      U     "MAL1S022Par".Par.FlagProcess2.Turning1WithoutSpraying;
      U     "MAL1S022Par".Par.FlagFunction_1.TurningStart;
      UN    "G205M".A_2611_MXZ41MA.Ma.StAdjusted; // target position turning reached
      FP    "MAL1S022Par".Par.FlagProcess2.StartFirstTurningFP;
      =     "MAL1S022Par".Par.FlagProcess2.StartFirstDosingFP;
      S     "MAL1S022Par".Par.FlagProcess2.StartFirstTurningRound;

      U     "MAL1S022Par".Par.FlagProcess2.StartFirstDosingFP;
      U     "MAL1S022Par".Par.FlagProcess2.StartFirstTurningFP;
      SPB   trn1;
      L     "MAL1S022Par".Par.ParIntMachine.ActualStep;
      T     "MAL1S022Par".Par.ParIntProcess.PrevStep1stTurn;
trn1: NOP   0;

      U     "G205M".A_2611_MXZ41MA.Ma.StAdjusted; // target position turning reached
      O(    ;
      L     "MAL1S022Par".ActTimeStepProcess.StepTimeActHourTotal; // Steptime in hours overall
      L     "MAL1S022Par".StepAct.StartTurningRound_1;
      >I    ;
      U(    ;
      O     "G205M".A_2611_MXZ41MA.Ma.OutAdjusted; // target position turning reached
      O(    ;
      UN    "G205M".A_2611_BZS46.StTrue; // stop fan side
      U     "G205M".A_2611_BZS44.StTrue; // stop discharge side
      U     "MAL1S022Par".Par.FlagFunction_1.TurningRight;
      )     ;
      O(    ;
      U     "G205M".A_2611_BZS46.StTrue; // stop fan side
      UN    "G205M".A_2611_BZS44.StTrue; // stop discharge side
      U     "MAL1S022Par".Par.FlagFunction_1.TurningLeft;
      )     ;
      )     ;
      )     ;
      O(    ;
      L     "MAL1S022Par".StepAct.StartTurningRound_1;
      L     0;
      <D    ; // negative, no turning 1
      )     ;
      U     "MAL1S022Par".Par.FlagProcess2.StartFirstTurningRound;
      R     "MAL1S022Par".Par.FlagProcess2.StartFirstTurningRound;
      R     "MAL1S022Par".Par.Switches1.StaOn08; // Turning1WithSpraying
      R     "MAL1S022Par".Par.Switches1.StaOn09; // Turning1WithDosing

// turning 2
      UN    "MAL1S022Par".Par.FlagProcess2.StartFirstTurningRound; // Unsinnige Rezeptwerte
      U(    ;
      L     1;
      L     "MAL1S022Par".StepAct.StartTurningRound_2;
      <>I   ;
      )     ;
      U(    ;
      O(    ; // Nach Rezept
      L     "MAL1S022Par".ActTimeStepProcess.StepTimeActHourTotal; // Steptime in hours overall
      L     "MAL1S022Par".StepAct.StartTurningRound_2;
      ==I   ;
      UN    "G205M".A_2611_MXZ41MA.Ma.StAdjusted; // target position turning reached
      )     ;
      O(    ; // Selbsthaltung
      L     "MAL1S022Par".ActTimeStepProcess.StepTimeActHourTotal; // Steptime in hours overall
      L     "MAL1S022Par".StepAct.StartTurningRound_2;
      <>I   ;
      U     "MAL1S022Par".Par.FlagProcess2.StartSecondTurningRound;
      )     ;
      )     ;
      S     "MAL1S022Par".Par.FlagProcess2.Turning2WithoutSpraying;
      S     "MAL1S022Par".Par.FlagFunction_1.TurningStart;
// turning 2 with spraying
      U(    ;
      L     1;
      L     "MAL1S022Par".StepAct.TurningWithSpraying_2;
      ==I   ;
      U(    ;
      L     "MAL1S022Par".Par.ParIntMachine.ActualStep;
      L     "MAL1S022Par".Par.ParIntProcess.PrevStep2ndTurn;
      ==I   ;
      )     ;
      )     ;
      O(    ;
      L     "MAL1S022Par".Par.ParIntMachine.ActualStep;
      L     "MAL1S022Par".Par.ParIntProcess.PrevStep2ndTurn;
      <>I   ;
      U     "MAL1S022Par".Par.Switches1.StaOn10; // Turning2WithSpraying
      )     ;
      U     "MAL1S022Par".Par.FlagProcess2.Turning2WithoutSpraying;
      S     "MAL1S022Par".Par.FlagProcess2.Turning2WithSpraying;
// turning 2 with spraying and GA3
      U(    ;
      L     1;
      L     "MAL1S022Par".StepAct.TurningWithDosing_2;
      ==I   ; // turning 2 with spraying and GA3 on
      U(    ;
      L     "MAL1S022Par".Par.ParIntMachine.ActualStep;
      L     "MAL1S022Par".Par.ParIntProcess.PrevStep2ndTurn;
      ==I   ;
      )     ;
      )     ;
      O(    ;
      L     "MAL1S022Par".Par.ParIntMachine.ActualStep;
      L     "MAL1S022Par".Par.ParIntProcess.PrevStep2ndTurn;
      <>I   ;
      U     "MAL1S022Par".Par.Switches1.StaOn11; // Turning2WithDosing
      )     ;
      U     "MAL1S022Par".Par.FlagProcess2.Turning2WithoutSpraying;
      S     "MAL1S022Par".Par.FlagProcess2.Turning2WithSpraying;
      S     "MAL1S022Par".Par.FlagProcess2.Turning2WithDosing;

      U     "MAL1S022Par".Par.FlagProcess2.Turning2WithoutSpraying;
      U     "MAL1S022Par".Par.FlagFunction_1.TurningStart;
      UN    "G205M".A_2611_MXZ41MA.Ma.StAdjusted; // target position turning reached
      FP    "MAL1S022Par".Par.FlagProcess2.StartSecondTurningFP;
      =     "MAL1S022Par".Par.FlagProcess2.StartSecondDosingFP;
      S     "MAL1S022Par".Par.FlagProcess2.StartSecondTurningRound;

      U     "MAL1S022Par".Par.FlagProcess2.StartSecondDosingFP;
      U     "MAL1S022Par".Par.FlagProcess2.StartSecondTurningFP;
      SPB   trn2;
      L     "MAL1S022Par".Par.ParIntMachine.ActualStep;
      T     "MAL1S022Par".Par.ParIntProcess.PrevStep2ndTurn;
trn2: NOP   0;

      U     "G205M".A_2611_MXZ41MA.Ma.StAdjusted; // target position turning reached
      O(    ;
      L     "MAL1S022Par".ActTimeStepProcess.StepTimeActHourTotal; // Steptime in hours overall
      L     "MAL1S022Par".StepAct.StartTurningRound_2;
      >I    ;
      U(    ;
      O     "G205M".A_2611_MXZ41MA.Ma.OutAdjusted; // target position turning reached
      O(    ;
      UN    "G205M".A_2611_BZS46.StTrue; // stop fan side
      U     "G205M".A_2611_BZS44.StTrue; // stop discharge side
      U     "MAL1S022Par".Par.FlagFunction_1.TurningRight;
      )     ;
      O(    ;
      U     "G205M".A_2611_BZS46.StTrue; // stop fan side
      UN    "G205M".A_2611_BZS44.StTrue; // stop discharge side
      U     "MAL1S022Par".Par.FlagFunction_1.TurningLeft;
      )     ;
      )     ;
      )     ;
      O(    ;
      L     "MAL1S022Par".StepAct.StartTurningRound_2;
      L     0;
      <D    ; // negative, no turning 2
      )     ;
      U     "MAL1S022Par".Par.FlagProcess2.StartSecondTurningRound;
      R     "MAL1S022Par".Par.FlagProcess2.StartSecondTurningRound;
      R     "MAL1S022Par".Par.Switches1.StaOn10; // Turning2WithSpraying
      R     "MAL1S022Par".Par.Switches1.StaOn11; // Turning2WithDosing

      L     3600;
      T     "MAL1S022Par".Par.ParIntMachine.TargetPosTravDriTurnRigt; // 360° = endposition turning right

// find turning direction spez. APU: right ==> forward, left ==> reverse
      U     "MAL1S022Par".Par.FlagGen.TurningStarted;
      O(    ;
      UN    "MAL1S022Par".Par.FlagProcess2.Turning1WithoutSpraying;
      UN    "MAL1S022Par".Par.FlagProcess2.Turning2WithoutSpraying;
      )     ;
      SPB   tuen;
      L     "MAL1S022Par".Par.ParIntMachine.TargetPosTravDriTurnRigt; // 360° = endposition turning right
      T     "G205M".A_2611_MXZ41MA.Ma.InPositionTarget; // target position turning

      U(    ;
      L     "G205M".A_2611_MXZ41MA.Ma.OutPositionAngle;
      L     1800;
      <I    ; // condition turning right (clockwise)
      )     ;
      O     "G205M".A_2611_BZS46.StTrue; // stop fan side
      UN    "G205M".A_2611_BZS44.StTrue; // stop discharge side
      S     "MAL1S022Par".Par.FlagFunction_1.TurningRight;
      S     "MAL1S022Par".Par.FlagGen.TurningStarted;
      SPB   E603;
      L     "MAL1S022Par".Par.ParIntMachine.TargetPosTravDriTurnLeft; // 0° = endposition turning left
      T     "G205M".A_2611_MXZ41MA.Ma.InPositionTarget; // target position turning

      U(    ;
      L     "G205M".A_2611_MXZ41MA.Ma.OutPositionAngle;
      L     1800;
      >=I   ; // condition turning left (counterclockwise)
      )     ;
      O     "G205M".A_2611_BZS44.StTrue; // stop discharge side
      UN    "G205M".A_2611_BZS46.StTrue; // stop fan side
      S     "MAL1S022Par".Par.FlagFunction_1.TurningLeft;
      S     "MAL1S022Par".Par.FlagGen.TurningStarted;
      SPB   E603;
tuen: NOP   0;

// reset turning right (clockwise)
      U     "MAL1S022Par".Par.FlagFunction_1.TurningRight;
      U(    ;
//      O     "G202M"._2111_MXZ41MA.Ma.StAdjusted    // target position turning reached
      O(    ;
      L     "G205M".A_2611_MXZ41MA.Ma.OutPositionAngle;
      L     "G205M".A_2611_MXZ41MA.Ma.Par.ParTolPosition;
      +I    ;
      L     "MAL1S022Par".Par.ParIntMachine.TargetPosTravDriTurnRigt;
      >=I   ;
      )     ;
      O     "G205M".A_2611_BZS44.StTrue; // stop discharge side
      )     ;
      R     "MAL1S022Par".Par.FlagFunction_1.TurningRight;
      R     "MAL1S022Par".Par.FlagFunction_1.TurningStart;

// reset turning left (counterclockwise)
      U     "MAL1S022Par".Par.FlagFunction_1.TurningLeft;
      U(    ;
//      O     "G202M"._2111_MXZ41MA.Ma.StAdjusted    // target position turning reached
      O(    ;
      L     "G205M".A_2611_MXZ41MA.Ma.OutPositionAngle;
      L     "G205M".A_2611_MXZ41MA.Ma.Par.ParTolPosition;
      -I    ;
      L     "MAL1S022Par".Par.ParIntMachine.TargetPosTravDriTurnLeft;
      <=I   ;
      )     ;
      O     "G205M".A_2611_BZS46.StTrue; // stop fan side
      )     ;
      R     "MAL1S022Par".Par.FlagFunction_1.TurningLeft;
      R     "MAL1S022Par".Par.FlagFunction_1.TurningStart;

// - Case of fast speed to protect a 2nd start during same hours as finsihed
      U     "MAL1S022Par".Par.FlagGen.TurningStarted;
      UN    "MAL1S022Par".Par.FlagProcess.ProcessEnd; // JV210808 to finish last turning
      UN    "MAL1S022StepValues".StartStep; // start step for average calculating
      U(    ;
      O(    ; // Nach Rezept
      L     "MAL1S022Par".ActTimeStepProcess.StepTimeActHourTotal; // Steptime in hours overall
      L     "MAL1S022Par".StepAct.StartTurningRound_1;
      <=I   ; // JV 250808
      UN    "MAL1S022Par".Par.FlagProcess2.StartFirstTurningRound; // JV 250808
      )     ;
      O(    ; // Nach Rezept
      L     "MAL1S022Par".ActTimeStepProcess.StepTimeActHourTotal; // Steptime in hours overall
      L     "MAL1S022Par".StepAct.StartTurningRound_2;
      <=I   ; // JV 250808
      UN    "MAL1S022Par".Par.FlagProcess2.StartSecondTurningRound; // JV 250808
      )     ;
      )     ;
      O(    ;
      UN    "G205M".A_2611_MXZ41MA.Ma.OutAdjusted; // target position turning reached
      UN    "MAL1S022Par".Par.FlagFunction_1.StepUnloading;
      )     ;
      SPB   e603;

// reset turning flag
      U     "MAL1S022Par".Par.FlagGen.TurningStarted;
      ON    "MAL1S022Par".Par.FlagProcess.ProcessActive;
      R     "MAL1S022Par".Par.FlagGen.TurningStarted;
      R     "MAL1S022Par".Par.FlagProcess2.Turning1WithoutSpraying;
      R     "MAL1S022Par".Par.FlagProcess2.Turning2WithoutSpraying;
      R     "MAL1S022Par".Par.FlagProcess2.Turning1WithSpraying;
      R     "MAL1S022Par".Par.FlagProcess2.Turning2WithSpraying;
      R     "MAL1S022Par".Par.FlagProcess2.Turning1WithDosing;
      R     "MAL1S022Par".Par.FlagProcess2.Turning2WithDosing;
      R     "MAL1S022Par".Par.FlagFunction_1.TurningStart;
      R     "MAL1S022Par".Par.FlagProcess2.StartFirstTurningRound; // JV 250808
      R     "MAL1S022Par".Par.FlagProcess2.StartSecondTurningRound; // JV 250808
      SET   ;
      R     "MAL1S022StepValues".StartStep; // start step for average calculating
e630: NOP   0;
      UN    "MAL1S022Par".Par.FlagProcess.ProcessActive;
      R     "MAL1S022Par".Par.FlagProcess2.StartFirstTurningRound;
      R     "MAL1S022Par".Par.FlagProcess2.StartSecondTurningRound;
      R     "MAL1S022Par".Par.Switches1.StaOn08; // Turning1WithSpraying
      R     "MAL1S022Par".Par.Switches1.StaOn09; // Turning1WithDosing
      R     "MAL1S022Par".Par.Switches1.StaOn10; // Turning2WithSpraying
      R     "MAL1S022Par".Par.Switches1.StaOn11; // Turning2WithDosing

      L     "G205M".A_2611_MXZ41MA.Ma.OutPositionAngle;
      T     "G205M".A_2611_MXZ41MA.Ma.OutPositionAngle;

      L     "G205M".A_2611_MXZ41MA.Ma.OutPositionRel;
      T     "G205M".A_2611_MXZ41MA.Ma.OutPositionRel;

e603: NOP   0;
E603: NOP   0;


NETWORK
TITLE =ASW_6040: Set fanspeed by delta-t
//Die Drehzahl des Ventilators wird zwischen dem Rezeptsollwert, als Untere
//Grenze, und 100% oder Rezeptsollwert, als obere Grenze, geregelt. Die Regelung
//erfolgt nach folgendem Prinzip:
//"Delta-T" ist die Differenz zwischen der Soll-Temperatur (Rezeptsollwert) unter
//der Horde und der gemessenen Ist-Temperatur über der Horde.
//Steigt die Ist-Temperatur über der Horde und "Delta-T" wird > als der Sollwert
//im Rezept, so wird die Drehzahl des Ventilators stufenweise erhöht. Maximale
//Drehzahl ist 100% oder Rezeptsollwert.
//Sinkt die Ist-Temperatur über der Horde und "Delta-T" wird < als der Sollwert
//im
//Rezept, so wird die Drehzahl des Ventilators stufenweise verringert. Minimale
//Drehzahl ist der Rezeptsollwert.
//Die Rampen (Stufen) werden durch den Technologen festgelegt und in Programmcode
//eingetragen. Es sind keine Rezeptsollwerte.
      NOP   0;
// recipe setpoint
      L     "MAL1S022Par".StepAct.SpeedVentilatorBasic;
      L     0;
      ==I   ; // no fan during turning
      SPB   e604; // JV040908
      L     "MAL1S022Par".Par.ProcessValue.StepTimeAct; // in ms
      L     L#1000; // in first secunde steptime
      >D    ;
      SPB   regu;
      SPA   Summ;
regu: NOP   0;

      U     "MAL1S022".ToASW.CmdModify;
      SPB   Summ;

// Setpoint
      L     "MAL1S022Par".StepAct.TemperaturAboveFloor;
      L     "MAL1S022Par".StepAct.TemperaturBelowFloor;
      -D    ;
      T     "MAL1S022Par".Par.ProcessValue.SetpointDeltaTempDint;
// actual value
      L     "G208M".A_2691_BTE02.OutValueUnits; //AIR TEMPERATURE ABOVE FLOOR
      L     "G208M".A_2691_BTE01.OutValueUnits; //AIR TEMPERATURE BELOW FLOOR
      -D    ;
      T     "MAL1S022Par".Par.ProcessValue.ActValueDeltaTempDint;
// flags to inc/dec
      L     "MAL1S022Par".Par.ProcessValue.SetpointDeltaTempDint;
      -D    ;
      T     "MAL1S022Par".Par.ProcessValue.ResultDeltaTemp;
      L     L#0;
      >D    ;
      =     "MAL1S022Par".Par.FlagProcess1.DeltaTempPlus;
      <D    ;
      =     "MAL1S022Par".Par.FlagProcess1.DeltaTempMinus;

      U     "MAL1S022Par".Par.FlagProcess1.DeltaTempPlus;
      U     "SYS_Scan0_Tick1min";
      SPBN  dec;
      L     "MAL1S022Par".Par.ParIntMachine.TargetSpeedGermFan;
      L     100; // linmit max
      >=I   ;
      SPB   dec;
      L     "MAL1S022Par".Par.ParIntMachine.TargetSpeedGermFan;
      L     1;
      +I    ;
      T     "MAL1S022Par".Par.ParIntMachine.TargetSpeedGermFan;
      SPA   e604;
dec:  NOP   0;
      U     "MAL1S022Par".Par.FlagProcess1.DeltaTempMinus;
      U     "SYS_Scan0_Tick1min";
      SPBN  e604;
      L     "MAL1S022Par".Par.ParIntMachine.TargetSpeedGermFan;
      L     "MAL1S022Par".StepAct.SpeedVentilatorBasic; // linmit min
      <=I   ;
      SPB   e604;
      L     "MAL1S022Par".Par.ParIntMachine.TargetSpeedGermFan;
      L     1;
      -I    ;
      T     "MAL1S022Par".Par.ParIntMachine.TargetSpeedGermFan;
      SPA   e604;

Summ: NOP   0;
      L     "MAL1S022Par".StepAct.SpeedVentilatorBasic;
      T     "MAL1S022Par".Par.ParIntMachine.TargetSpeedGermFan;
      U     "MAL1S022Par".Par.FlagProcess.ProcessEnd; // JV030908
      UN    "MAL1S022".PCRead.Step.StEmptying;
      UN    "MAL1S022".PCRead.Step.StEmptied;
      SPBN  e604;
      L     "MAL1S022Par".Par.ParIntProcess.SavedTargetSpeedGermFan;
      T     "MAL1S022Par".Par.ParIntMachine.TargetSpeedGermFan;
e604: NOP   0;
// store actual setpoint
      U     "MAL1S022Par".Par.FlagProcess.ProcessActive;
      U(    ;
      L     "MAL1S022Par".StepAct.SpeedVentilatorBasic;
      L     0; // setpoint recipe > 0
      >I    ;
      )     ;
      SPBN  E604;
      L     "MAL1S022Par".StepAct.SpeedVentilatorBasic;
      T     "MAL1S022Par".Par.ParIntProcess.SavedTargetSpeedGermFan;
E604: NOP   0;

NETWORK
TITLE =ASW_6050: Position waste air
//Der Betriebsart Sommerbetrieb/Winterbetrieb wird durch den Bediener per Rezept
//bestimmt.
//Wird die Kühlung im Rezept angewählt, so erfolgt die Umschaltung AUF
//Sommerbetrieb. Die Frischluftklappe wird nach dem Rezeptsollwert gestellt.
//Es erfolgt keine Regelung.
//Wird die Kühlung im Rezept abgewählt, so erfolgt die Umschaltung AUF
//Winterbetrieb. Die Frischluftklappe wird zuerst nach dem Rezeptsollwert
//gestellt. Der Rezeptsollwert ist die untere Grenze für die Regelung.
//Wird die Soll-Temperatur unter der Horde von Kühl- Heizanlage nicht eingehalten
//-Temperatur zu hoch und der Schaltpunkt überschritten, so wird die
//Frischluftklappe stufenweise geöffnet.
//Maximalwert ist 100%.
//Wird die Soll-Temperatur unter der Horde von Kühl- Heizanlage nicht eingehalten
//-Temperatur zu niedrig und der Schaltpunkt unterschritten, so wird die
//Frischluftklappe stufenweise geschlossen.
//Minimalwert ist der Rezeptsollwert.
      NOP   0;
// setpoint waste air                    = 100% - setpoint fresh air
      L     100;
      L     "MAL1S022Par".StepAct.PosFreshAirFlapBasic;
      -I    ;
      T     "MAL1S022Par".StepAct.PosWasteAirFlapBasic;

// setpoint limit maximal position fresh air
      L     100;
      T     "MAL1S022Par".StepAct.PosFreshAirFlapMax; // limit max
      L     L#10; // 1,0°
      T     "MAL1S022Par".StepAct.DeltaTempSwitchpointAir;

// recipe setpoint
      L     "MAL1S022Par".Par.ProcessValue.StepTimeAct; // in ms
      L     L#1000; // in first secunde steptime
      >D    ;
      SPB   Reg;
      SPA   summ;
Reg:  NOP   0;

// Cooling or heating from cooling defive active --> no flap regulation!
//      U     "ENG_RemarkFlag"
//      U     "ComDB_Cooling".Ma.ACK.ActivFlag.Cool.Germinating_1_Started // Internal or external coooling is running
//      O     "MAL1S017".ToASW.CmdModify
//      SPB   summ

//Conditions to activate cooling -- With flap regulation
      U(    ;
      L     1;
      L     "MAL1S022Par".StepAct.Cooling; // On/Off
      ==I   ; // Cooling on
      U     "MAL1S022Par".Par.FlagProcess.ProcessActive;
      )     ;
      U     "G210M".A_2660_MXZ01.StStartedFwd;
      U     "G210M".A_2660_MXZ02.StStartedFwd;
      U(    ;
      L     "G269M".A_3191_BTE11.OutValueUnits; //WET BULB TEMPERATURE OUTSIDE
      L     20; // 2,0°C Hysteresis
      -D    ;
      L     "MAL1S022Par".StepAct.TemperaturBelowFloor; //SET POINT TEMPERATURE RECIPE
      >=D   ;
      )     ;
      U(    ;
      L     "G208M".A_2691_BTE01.OutValueUnits; //AIR TEMPERATURE BELOW FLOOR GM2
      L     10; // 1,0°C Hysteresis
      -D    ;
      L     "MAL1S022Par".StepAct.TemperaturBelowFloor; //SET POINT TEMPERATURE RECIPE
      >=D   ;
      )     ;
      U(    ;
      L     "G208M".A_2691_BTE02.OutValueUnits; //AIR TEMPERATURE ABOVE FLOOR GM2
      L     20; // 2,0°C Hysteresis
      -D    ;
      L     "MAL1S022Par".StepAct.TemperaturBelowFloor; //SET POINT TEMPERATURE RECIPE
      >=D   ;
      )     ;
      S     "MAL1S022Par".Par.FlagProcess.Cooling_Activ;

      U(    ;
      L     0;
      L     "MAL1S022Par".StepAct.Cooling; // On/Off
      ==I   ; // Cooling off
      )     ;
      ON    "G210M".A_2660_MXZ01.StStartedFwd;
      ON    "G210M".A_2660_MXZ02.StStartedFwd;
      O(    ;
      L     "G269M".A_3191_BTE11.OutValueUnits; //WET BULB TEMPERATURE OUTSIDE
      L     10; // 1,0°C Hysteresis
      +D    ;
      L     "MAL1S022Par".StepAct.TemperaturBelowFloor; //SET POINT TEMPERATURE RECIPE
      <D    ;
      )     ;
      O(    ;
      L     "G208M".A_2691_BTE02.OutValueUnits; //AIR TEMPERATURE ABOVE FLOOR GM1
      L     10; // 1,0°C Hysteresis
      +D    ;
      L     "MAL1S022Par".StepAct.TemperaturBelowFloor; //SET POINT TEMPERATURE RECIPE
      <D    ;
      )     ;
      R     "MAL1S022Par".Par.FlagProcess.Cooling_Activ;

      U     "MAL1S022Par".Par.FlagProcess.Cooling_Activ;
      SPB   summ;

// Check the minimum opening of fresh air louver
      U(    ;
      L     "MAL1S022Par".Par.ParIntMachine.TargetPosFreshAir;
      L     "MAL1S022Par".StepAct.PosFreshAirFlapBasic;
      <I    ;
      )     ;
      SPBN  modi;
      L     "MAL1S022Par".StepAct.PosFreshAirFlapBasic; //Basic position %
      T     "MAL1S022Par".Par.ParIntMachine.TargetPosFreshAir;
modi: NOP   0;

//-Recipe modify-
      U(    ; // Nach gesundem Menschenverstand
      L     "MAL1S022Par".StepAct.PosFreshAirFlapBasic;
      L     "MAL1S022Par".Par.ParIntMachine.TargetPosFreshAir;
      >I    ;
      U     "MAL1S022Par".Par.FlagProcess1.FreshAirFlapOPEN;
      )     ;
      O(    ; // Nach gesundem Menschenverstand
      L     "MAL1S022Par".StepAct.PosFreshAirFlapBasic;
      L     "MAL1S022Par".Par.ParIntMachine.TargetPosFreshAir;
      <I    ;
      U     "MAL1S022Par".Par.FlagProcess1.FreshAirFlapCLOSE;
      )     ;
      O(    ; // Nach gesundem Menschenverstand
      L     "MAL1S022Par".StepAct.PosFreshAirFlapBasic;
      L     "MAL1S022Par".Par.ParIntMachine.TargetPosFreshAir;
      <>I   ;
      UN    "MAL1S022Par".Par.FlagProcess1.FreshAirFlapOPEN;
      UN    "MAL1S022Par".Par.FlagProcess1.FreshAirFlapCLOSE;
      )     ;
      O(    ; // 1. Versuch den Technologen ruhig stellen
      L     "MAL1S022Par".StepAct.PosFreshAirFlapBasic;
      L     "MAL1S022Par".Par.ParIntProcess.SavedTargetPosFreshAir;
      <>I   ;
      )     ;
      U     "MAL1S022".ToASW.CmdModify;
      SPB   summ;
//      L     "G168M".A_2491_BTE01.OutValueUnits    //AIR TEMPERATURE BELOW FLOOR
//      L     L#10                        // von xx,xx°C AUF xx,x°C
//      /D
//      L     "MAL1S017Par".StepAct.TemperaturBelowFloor
//      -D
//      L     "MAL1S017Par".StepAct.DeltaTempSwitchpointAir
//      >D
//      =     "MAL1S017Par".Par.FlagProcess1.FreshAirFlapOPEN

//      L     "G128M".A_2191_BTE01.OutValueUnits    //AIR TEMPERATURE BELOW FLOOR
//      L     L#10                        // von xxx,xx°C AUF xxx,x°C
//      /D
//      L     "MAL1S017Par".StepAct.TemperaturBelowFloor
//      TAK
//      -D
//      L     "MAL1S017Par".StepAct.DeltaTempSwitchpointAir
//      >D
//      =     "MAL1S017Par".Par.FlagProcess1.FreshAirFlapCLOSE
      U(    ;
      L     "G208M".A_2691_BTE01.OutValueUnits; //AIR TEMPERATURE BELOW FLOOR GM1
      L     "MAL1S022Par".StepAct.TemperaturBelowFloor; //SET POINT TEMPERATURE RECIPE
      <D    ;
      )     ;
      U(    ;
      L     "G269M".A_3191_BTE11.OutValueUnits; //WET BULB TEMPERATURE OUTSIDE
      L     "G208M".A_2691_BTE02.OutValueUnits; //AIR TEMPERATURE ABOVE FLOOR GM1
      >D    ;
      )     ;
      O     ;
      U(    ;
      L     "G208M".A_2691_BTE01.OutValueUnits; //AIR TEMPERATURE BELOW FLOOR GM1
      L     "MAL1S022Par".StepAct.TemperaturBelowFloor; //SET POINT TEMPERATURE RECIPE
      >D    ;
      )     ;
      U(    ;
      L     "G269M".A_3191_BTE11.OutValueUnits; //WET BULB TEMPERATURE OUTSIDE
      L     "G208M".A_2691_BTE01.OutValueUnits; //AIR TEMPERATURE BELOW FLOOR GM1
      <D    ;
      )     ;
      =     "MAL1S022Par".Par.FlagProcess1.FreshAirFlapOPEN;

      U(    ;
      L     "G208M".A_2691_BTE01.OutValueUnits; //AIR TEMPERATURE BELOW FLOOR GM1
      L     "MAL1S022Par".StepAct.TemperaturBelowFloor; //SET POINT TEMPERATURE RECIPE
      <D    ;
      )     ;
      U(    ;
      L     "G269M".A_3191_BTE11.OutValueUnits; //WET BULB TEMPERATURE OUTSIDE
      L     "G208M".A_2691_BTE02.OutValueUnits; //AIR TEMPERATURE ABOVE FLOOR GM1
      <D    ;
      )     ;
      =     "MAL1S022Par".Par.FlagProcess1.FreshAirFlapCLOSE;

      U     "MAL1S022Par".Par.FlagProcess1.FreshAirFlapOPEN;
      U     "SYS_Scan0_Tick1min";
      SPBN  dez;
      L     "MAL1S022Par".Par.ParIntMachine.TargetPosWasteAir;
      L     100; // limit max
      >=I   ;
      SPB   dez;
      L     "MAL1S022Par".Par.ParIntMachine.TargetPosWasteAir;
      L     1;
      +I    ;
      T     "MAL1S022Par".Par.ParIntMachine.TargetPosWasteAir;
      SPA   e605;
dez:  NOP   0;
      U     "MAL1S022Par".Par.FlagProcess1.FreshAirFlapCLOSE;
      U     "SYS_Scan0_Tick1min";
      SPBN  e605;
      L     "MAL1S022Par".Par.ParIntMachine.TargetPosWasteAir;
      L     "MAL1S022Par".StepAct.PosFreshAirFlapBasic; // limit min
      <=I   ;
      SPB   e605;
      L     "MAL1S022Par".Par.ParIntMachine.TargetPosWasteAir;
      L     1;
      -I    ;
      T     "MAL1S022Par".Par.ParIntMachine.TargetPosWasteAir;
      SPA   e605;

summ: NOP   0;
      U     "G269M".read_3191;
      SPBN  bypa;
      U(    ;
      L     "G208M".A_2691_BTE02.OutValueUnits; //AIR TEMPERATURE ABOVE FLOOR GM1
      L     10; // 1,0°C Hysteresis
      -D    ;
      L     "G269M".A_3191_BTE11.OutValueUnits; //WET BULB TEMPERATURE OUTSIDE
      >=D   ;
      )     ;
      SPB   tar1;
      U(    ;
      L     "G208M".A_2691_BTE02.OutValueUnits; //AIR TEMPERATURE ABOVE FLOOR GM1
      L     10; // 1,0°C Hysteresis
      +D    ;
      L     "G269M".A_3191_BTE11.OutValueUnits; //WET BULB TEMPERATURE OUTSIDE
      <=D   ;
      )     ;
      SPB   tar0;
      SPA   bypa;
tar1: L     100; //open fresh air 100%
      T     "MAL1S022Par".Par.ParIntMachine.TargetPosFreshAir;
      SPA   bypa;
tar0: L     "MAL1S022Par".StepAct.PosFreshAirFlapBasic; //close fresh air to Basic position %
      T     "MAL1S022Par".Par.ParIntMachine.TargetPosFreshAir;
bypa: NOP   0;
//************************************************************************
      U     "MAL1S022Par".Par.FlagProcess.ProcessEnd; // JV030908
      UN    "MAL1S022".PCRead.Step.StEmptying;
      UN    "MAL1S022".PCRead.Step.StEmptied; // JV030908
      SPBN  e605;
      L     "MAL1S022Par".Par.ParIntProcess.SavedTargetPosFreshAir;
      T     "MAL1S022Par".Par.ParIntMachine.TargetPosFreshAir;
e605: NOP   0;
      L     100;
      L     "MAL1S022Par".Par.ParIntMachine.TargetPosFreshAir;
      -I    ;
      T     "MAL1S022Par".Par.ParIntMachine.TargetPosWasteAir;
// store actual setpoint
      U     "MAL1S022Par".Par.FlagProcess.ProcessActive;
      U(    ;
      L     "MAL1S022Par".StepAct.PosFreshAirFlapBasic;
      L     0; // setpoint recipe > 0
      >I    ;
      )     ;
      SPBN  E605;
      L     "MAL1S022Par".StepAct.PosFreshAirFlapBasic;
      T     "MAL1S022Par".Par.ParIntProcess.SavedTargetPosFreshAir;
E605: NOP   0;

NETWORK
TITLE =ASW_6080: Processtime Germinating
//      CALL  "SSA_MH_ProcessTime_Fct" , DB1017
//       InfDataReady :="MAL1S017".ToASW.InfDataReady
//       ProzessActive:="MAL1S017Par".Par.FlagProcess.ProcessActive
//       InStartTime  :="MAL1S017Par".Prozesstime.Starttime
//       OutStartTime :="MAL1S017Par".Prozesstime.Starttime
//       ProcessTime  :="MAL1S017Par".Prozesstime
//
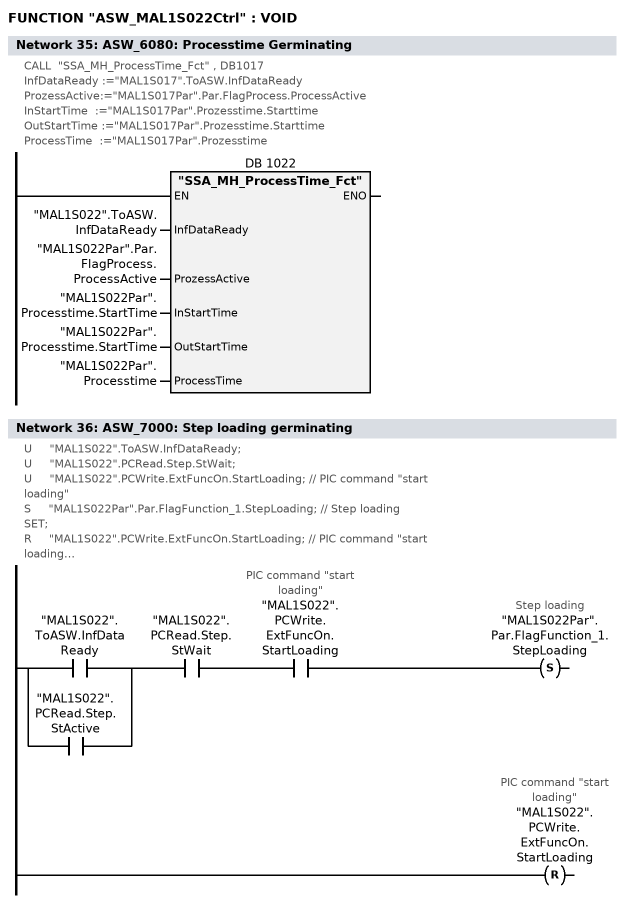
      CALL "SSA_MH_ProcessTime_Fct" , DB  1022 (
           InfDataReady             := "MAL1S022".ToASW.InfDataReady,
           ProzessActive            := "MAL1S022Par".Par.FlagProcess.ProcessActive,
           InStartTime              := "MAL1S022Par".Processtime.StartTime,
           OutStartTime             := "MAL1S022Par".Processtime.StartTime,
           ProcessTime              := "MAL1S022Par".Processtime);

NETWORK
TITLE =ASW_7000: Step loading germinating
//      U     "MAL1S022".ToASW.InfDataReady;
//      U     "MAL1S022".PCRead.Step.StWait;
//      U     "MAL1S022".PCWrite.ExtFuncOn.StartLoading; // PIC command "start
//loading"
//      S     "MAL1S022Par".Par.FlagFunction_1.StepLoading; // Step loading
//      SET;
//      R     "MAL1S022".PCWrite.ExtFuncOn.StartLoading; // PIC command "start
//loading"
////
//
//      L     WinCoS_BIW01_09PLC1BIW01_02.Ma.OutPositionAngle;
//      L     3600; // 360,0°
//      >=I   ;
//      U     "MAL1S022".ToASW.InfDataReady;
//      U     "MAL1S022".PCRead.Step.StActive;
//      U     "MAL1S022Par".Par.FlagFunction_1.StepLoading; // Step loading
//      =     "MAL1S022Par".Par.FlagFunction_1.LoadFirstPartEnd;
//
//      U     "MAL1S022".ToASW.InfDataReady;
//      U     "MAL1S022".PCRead.Step.StActive;
//      U     "MAL1S022Par".Par.FlagFunction_1.StepLoading; // Step loading
//      SPBN  E700;
//      L     "MAL1S022Par".RecipeHeader.Loading.LiftingPositionRound_1;
//      T     "MAL1S022Par".Par.ParIntProcess.NextLevelLoading; // next level
//
//      U(    ;
//      L     WinCoS_BIW01_09PLC1BIW01_02.Ma.OutPositionAngle;
//      L     "MAL1S022Par".Par.ParIntProcess.NextLevelLoading; // next level
//      >=I   ;
//      )     ;
//      O     "MAL1S022Par".Par.FlagMachine_0.Speed2ndRound;
//      SPB   Rnd2;
//      L     "MAL1S022Par".RecipeHeader.Loading.LoadingLevelRound_1;
//      T     "MAL1S022Par".Par.MachineValue.SOLLWERT_HUBZUG1_HOEHE;
//      T     "MAL1S022Par".Par.MachineValue.SOLLWERT_HUBZUG2_HOEHE;
//
//      L     "MAL1S022Par".RecipeHeader.Loading.LoadingSpeed_1;
//      T     "MAL1S022Par".Par.MachineValue.SollwertFahrantrieb;
//
//      SPA   Rnd1;
//Rnd2: NOP   0;
//      L     "MAL1S022Par".RecipeHeader.Loading.LoadingLevelRound_2;
//      T     "MAL1S022Par".Par.MachineValue.SOLLWERT_HUBZUG1_HOEHE;
//      T     "MAL1S022Par".Par.MachineValue.SOLLWERT_HUBZUG2_HOEHE;
//      L     10;
//      T     WinCoS_BIW01_09PLC1BIW01_02.Ma.Par.ParTolPosition;
//
//      L     15; // 15Hz = Wendegeschwindigkeit
//      T     "MAL1S022Par".Par.MachineValue.SollwertFahrantrieb;
//
//// Sicherheitsbit; damit bei manueller Rückwärtsfahrt über die 346°-Marke,
//nicht mit Loading Speed_0 durch den gefüllten KK gefahren wird!!
//      SET   ;
//      S     "MAL1S022Par".Par.FlagMachine_0.Speed2ndRound;
//
//Rnd1: NOP   0;
//      U  M 50.0;
//      =  M 50.0;
//      L     "MAL1S022Par".Par.ParIntMachine.TargetPosTravDriveLoad; // 450 =
//endposition loading
//      T     WinCoS_BIW01_09PLC1BIW01_02.Ma.InPositionTarget;
//E700: NOP   0;




      U     "MAL1S022".ToASW.InfDataReady;
      O     "MAL1S022".PCRead.Step.StActive;
      U     "MAL1S022".PCRead.Step.StWait;
      U     "MAL1S022".PCWrite.ExtFuncOn.StartLoading; // PIC command "start loading"
      S     "MAL1S022Par".Par.FlagFunction_1.StepLoading; // Step loading
      SET   ;
      R     "MAL1S022".PCWrite.ExtFuncOn.StartLoading; // PIC command "start loading"
//
      NOP   0;


NETWORK
TITLE =Sub 7010: Germination loading finished
//      U     "MAL1S022".ToASW.InfDataReady;
//      U     "MAL1S022".PCRead.Step.StActive;
//
//      UN    "MAL1S022".ToASW.InfSameJobPrevSec;
//      UN    "MAL1S022".PCRead.Step.StEmptying; // steep 1
//      U     "MAL1S022".PCWrite.ExtFuncOn.FinishLoading; // PIC command "finish l
//oading"
//      U     "MAL1S022Par".Par.FlagFunction_1.StepLoading; // Step loading
//      S     "MAL1S022Par".Par.FlagFunction_1.FinishLoading; // loading is
//finished start process germinating
//      R     "MAL1S022Par".Par.FlagFunction_1.StepLoading; // Step loading
//
//      U     "MAL1S022".PCWrite.ExtFuncOn.FinishLoading; // PIC command "finish
//loading"
//      R     "MAL1S022".PCWrite.ExtFuncOn.FinishLoading; // PIC command "finish
//loading"
//
//      U     "MAL1S022Par".Par.FlagFunction_1.StepLoading; // Step loading
//      UN    "MAL1S022Par".Par.FlagFunction_1.FinishLoading; // loading is
//finished start process germinating
//      SPBN  save;
//      L     WinCoS_BIW01_09PLC1BIW01_02.Ma.OutPositionLeft;
//      L     WinCoS_BIW01_09PLC1BIW01_02.Ma.OutPositionRight;
//      +I    ;
//      L     2;
//      /I    ;
//      T     "MAL1S022Par".Par.ParIntMachine.LastLoadingLevel; // saved loading
//value
//save: NOP   0;
//
//      U     "MAL1S022".PCRead.Step.StReady;
//      O     "MAL1S022".PCRead.Step.StActive;
//      U     "MAL1S022Par".Par.FlagFunction_1.FinishLoading; // loading is
//finished start process germinating
//      UN     "MAL1S022Par".Par.FlagFunction_1.StepLoading; // Step loading
//      R     "MAL1S022Par".Par.FlagMachine_0.Speed2ndRound;
//fin:  NOP   0;
//E701: NOP   0;





// U SPS geht in Stopp, weil DBW70=0 und DB0 gibt es nicht.
// Also, es ist schon grobe Fahrlässigkeit.
      L     "MAL1S022".ToSSW.InPrevSecDB;
      L     0;
      <>I   ;
      SPB   Voss;
      L     801;
      T     "MAL1S022".ToSSW.InPrevSecDB;
Voss: NOP   0;

      U     "MAL1S022".ToASW.InfDataReady;
      U     "MAL1S022".PCRead.Step.StActive;
//      UN    "MAL1S022".ToASW.InfSameJobPrevSec
//      U(
//      L     "MAL1S022".ToSSW.InPrevSecDB
//      T     #tmpInt
//      AUF   DB [#tmpInt]                // previous section is
//      U     DBX  111.5                  // emptied
//      O     DBX  111.6                  // idling
//      O     DBX  111.0                  // passive
//      ON    "MAL1S022".ToASW.InfSameBatchPrevSec    //dyk 081027 Steeping has new job but operator has not pushed "Finish loading"
//      )
      UN    "MAL1S022".PCRead.Step.StEmptying; //
      U     "MAL1S022".PCWrite.ExtFuncOn.FinishLoading; // PIC command "finish loading"
      U     "MAL1S022Par".Par.FlagFunction_1.StepLoading; // Step loading
      O(    ;
      UN    "MAL1S022".SecNom.Par1On.Cmd01; // With Loading
      UN    "MAL1S022".ToASW.InfSameBatchPrevSec;
      U     "MAL1S022".ToASW.InfDataReady;
      U     "MAL1S022".PCRead.Step.StActive;
      )     ;
      S     "MAL1S022Par".Par.FlagFunction_1.FinishLoading; // loading is finished start process germinating
      R     "MAL1S022Par".Par.FlagFunction_1.StepLoading; // Step loading

      U     "MAL1S022".PCWrite.ExtFuncOn.FinishLoading; // PIC command "finish loading"
      R     "MAL1S022".PCWrite.ExtFuncOn.FinishLoading; // PIC command "finish loading"


      U     "MAL1S022".PCRead.Step.StReady;
      O     "MAL1S022".PCRead.Step.StActive;
      U     "MAL1S022Par".Par.FlagFunction_1.FinishLoading; // loading is finished start process germinating
      UN    "MAL1S022Par".Par.FlagFunction_1.StepLoading; // Step loading
      R     "MAL1S022Par".Par.FlagMachine_0.Speed2ndRound;
      NOP   0;
      NOP   0;


NETWORK
TITLE =ASW_8000:  Step unloading germination



      U     "MAL1S022".ToASW.InfDataReady;
      U     "MAL1S022".PCRead.Step.StEmptying;
      U     "MAL1S022".ToASW.InfSameJobNextSec;
      UN    "MAL1S022Par".Par.FlagFunction_1.StepUnloading; // Step unloading
      UN    "MAL1S022Par".Par.FlagFunction_1.FinishUnloading;
      U     "MAL1S022Par".Par.FlagMachine_0.CouplingDischargFinished;
      U     "MAL1S022Par".Par.FlagMachine_0.WallUnCoupled;
      S     "MAL1S022Par".Par.FlagFunction_1.StepUnloading; // Step unloading

      U     "MAL1S022Par".Par.FlagFunction_1.StepUnloading; // Step unloading
      U     "MAL1S022Par".Par.FlagFunction_1.UnloadingStarted;
      U     "MAL1S022".ToASW.spare34; // infNextSectionFeeding
      =     "MAL1S022Par".Par.FlagFunction_0.InfReleaseUnloading; // from kiln

      U     "MAL1S022Par".Par.FlagFunction_1.StepUnloading; // Step unloading
      UN    "MAL1S022Par".Par.FlagFunction_1.UnloadingStarted;
      U     "G202M".A_2615_BZS22.StFalse; // backwall is not in down pos
      U     "G202M".A_2615_BZS23.StTrue; // backwall is in up pos  // JV030908
      U     "G207M".A_2611_KCL01I5.StTrue; // pushbutton drive fast fwd
      S     "MAL1S022Par".Par.FlagFunction_1.UnloadingStarted;
      FP    "MAL1S022Par".Par.FlagFunction_0.FlagUnloadingStartedFP; // JV030908
      =     "MAL1S022Par".Par.FlagFunction_0.ImpulseUnloadingStarted; // JV030908

      UN    "MAL1S022Par".Par.FlagFunction_1.UnloadingStarted;
      O     "MAL1S022Par".Par.FlagFunction_1.StepCleaning; // Step cleaning
      O     "MAL1S022Par".Par.FlagFunction_1.FinishCleaning;
      SPB   EN38;
      L     3600;
      T     "G205M".A_2611_MXZ41MA.Ma.InPositionTarget; // target position unloading
      L     "MAL1S022Par".RecipeHeader.Unloading.UnLoadingSpeed_2; // JV 290808
      T     "MAL1S022Par".Par.ParIntProcess.CopyLoadindSpeed2; // JV 290808
EN38: NOP   0;




NETWORK
TITLE =ASW_8010:  Step unloading finished



// Verweilzeit auf dem Endschalter  =A_2111_BZS44.StTrue --> stop discharge side
      L     S5T#10M; // Verweilzeit auf dem Endschalter
      U     "G205M".A_2611_BZS44.StTrue; // stop discharge side
      U     "G204M".A_2615_BZS42.StTrue;
      SE    T    122;
//************************************************************************************************

      U     "MAL1S022".ToASW.InfDataReady;
      U     "MAL1S022".PCRead.Step.StEmptying;
      U     "MAL1S022".ToASW.InfSameJobNextSec;
      U     "MAL1S022Par".Par.FlagFunction_1.StepUnloading; // Step unloading
      UN    "MAL1S022Par".Par.FlagFunction_1.FinishUnloading;
      U     "MAL1S022Par".Par.FlagFunction_1.StepUnloading; // Step unloading
      U     "MAL1S022Par".Par.FlagFunction_1.UnloadingStarted;
      U     T    122; // Verweilzeit auf dem Endschalter ist abgelaufen
//------------ Confirmation is necessary to finish unloading **********************
      U(    ;
      L     "G205M".A_2611_MXZ41MA.Ma.OutPositionRel;
      L     950; //95%
      >I    ;
      )     ;
//      U     "MAL1S022".PCWrite.ExtFuncOn.FinishCleanSurface    // PIC command "Finish Unloading"
//************************************************************************************************
      R     "MAL1S022Par".Par.FlagFunction_1.StepUnloading; // Step unloading
      S     "MAL1S022Par".Par.FlagFunction_1.FinishUnloading;
      S     "MAL1S022Par".Par.FlagMachine_0.CmdTurnRevAfterUnloading;
      UN    "MAL1S022Par".Par.FlagMachine_0.CmdTurnRevAfterUnloading;
      SPB   EN39;
      L     3399;
      T     "G205M".A_2611_MXZ41MA.Ma.InPositionTarget; // target position
EN39: NOP   0;

      SET   ;
      R     "MAL1S022".PCWrite.ExtFuncOn.FinishCleanSurface; // PIC command "Finish Unloading"




NETWORK
TITLE =ASW_9000: Step cleaning germination box
//
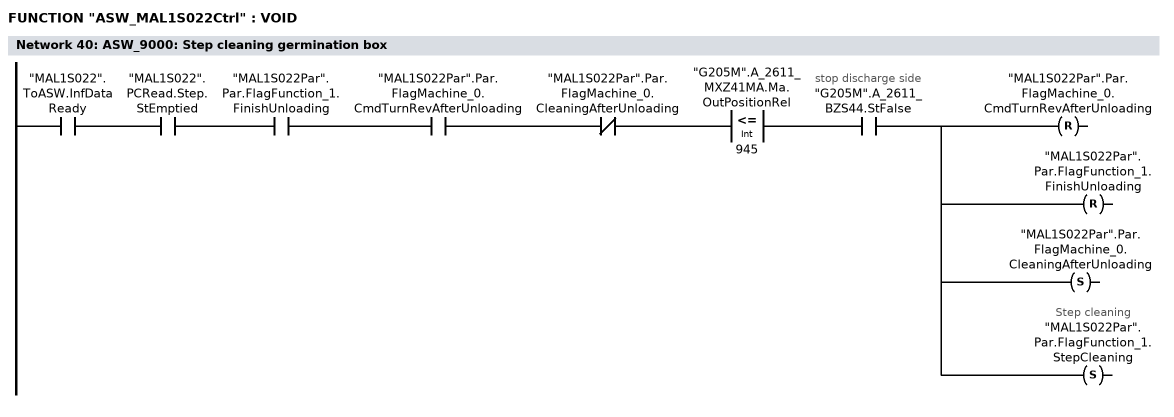

      U     "MAL1S022".ToASW.InfDataReady;
      U     "MAL1S022".PCRead.Step.StEmptied;
      U     "MAL1S022Par".Par.FlagFunction_1.FinishUnloading;
      U     "MAL1S022Par".Par.FlagMachine_0.CmdTurnRevAfterUnloading;
      UN    "MAL1S022Par".Par.FlagMachine_0.CleaningAfterUnloading;
      U(    ;
      L     "G205M".A_2611_MXZ41MA.Ma.OutPositionRel;
      L     945;
      <=I   ; // cleaning pos
      )     ;
      U     "G205M".A_2611_BZS44.StFalse; // stop discharge side
      R     "MAL1S022Par".Par.FlagMachine_0.CmdTurnRevAfterUnloading;
      R     "MAL1S022Par".Par.FlagFunction_1.FinishUnloading;
      S     "MAL1S022Par".Par.FlagMachine_0.CleaningAfterUnloading;
      S     "MAL1S022Par".Par.FlagFunction_1.StepCleaning; // Step cleaning

NETWORK
TITLE =ASW_9010: Cleaning Germination box finished
//



      U     "MAL1S022".ToASW.InfDataReady;
      U     "MAL1S022".PCRead.Step.StEmptied;
      U     "MAL1S022Par".Par.FlagFunction_1.StepCleaning; // Step cleaning
      U     "G205M".A_2611_BZS44.StFalse; // stop discharge side
      U(    ;
      O     "MAL1S022".PCWrite.ExtFuncOn.FinishCleaning; // PIC command "cleaning finished"
      O     "G207M".A_2611_KCL01I4.InpTrue; // pushbutton "drive rev"
      )     ;
      R     "MAL1S022Par".Par.FlagMachine_0.CleaningAfterUnloading;
      R     "MAL1S022Par".Par.FlagFunction_1.StepCleaning; // Step cleaning
      S     "MAL1S022Par".Par.FlagFunction_1.FinishCleaning;

      SET   ;
      R     "MAL1S022".PCWrite.ExtFuncOn.FinishCleaning; // PIC command "cleaning finished"

      U     "MAL1S022".PCRead.Step.StIdling;
      U     "G205M".A_2611_BZS46.StTrue; // stop fan side (home pos)
      U(    ; //dyk 081031 50 pulses
      L     "G205M".A_2611_MXZ41MA.IncCounter.InpActCount;
      L     50;
      <I    ;
      )     ;
      R     "MAL1S022Par".Par.FlagFunction_1.FinishCleaning;

      UN    "MAL1S022Par".Par.FlagFunction_1.FinishCleaning;
      SPB   EN41;
      L     0;
      T     "G205M".A_2611_MXZ41MA.Ma.InPositionTarget; // target position
//MW 2008.10.24
      L     "MAL1S022Par".RecipeHeader.Unloading.UnLoadingSpeed_2;
      T     "MAL1S022Par".Par.ParIntProcess.CopyLoadindSpeed2;
EN41: NOP   0;


NETWORK
TITLE =ASW_9080: Send section date to PIC after germination

      AUF   "MAL1S022";
      U     "MAL1S022".PCRead.Step.StEmptying;
      FP    "MAL1S022Par".Par.FlagProcess.FP_SendResultToPIC;
      SPBN  E908;
//

E908: NOP   0;
NETWORK
TITLE =ASW_10000: ILO functions

      U     "MAL1S022".SecAc.Sta1On.Inf08;
      =     "MAL1S022".Gr.All.Spare04;

// reset ILO with start unloading   JV080908    special on SALADIN BOXES
      U     "MAL1S022Par".Par.FlagFunction_0.ImpulseUnloadingStarted; // JV030908
      R     "MAL1S022".SecAc.Sta1On.Inf08;

//- Little help for PIC-People
      U     "MAL1S022".SecAc.Sta1On.Inf08;
      SPB   RSM;
      L     0;
      T     "MAL1S022Par".Ilo.Code_ILO_Funktion0; // FCM 19 LINE 1 SEC 19  GERM 6
RSM:  NOP   0;
//- Combination OLD and NEW ---
      U     "MAL1S022".SecAc.Sta1On.Inf08;
      SPBN  IFM;
      L     "MAL1S022Par".Ilo.ILOMode;
      L     100;
      *I    ;
      T     "MAL1S022Par".Ilo.Code_ILO_Funktion0;
IFM:  NOP   0;

//  no ILO-mode >> cmd manual off to all used groups and reset all flags
      U     "MAL1S022".SecAc.Sta1On.Inf08;
      FN    DB909.DBX 3692.0;
//      S     DB909.DBX 3006.0            // (ManOff)
//      R     DB909.DBX 3014.0
//      R     DB909.DBX 3018.1
//  Gr-cmd manual OFF
      S     "G202M".Gr.CmdManualOff; // LIFTING DEVICE  GERM 6
      S     "G203M".Gr.CmdManualOff; // COUPLING DEVICE TURNER  GERM 6
      S     "G204M".Gr.CmdManualOff; // COUPLING DEVICE WALL  GERM 6
      S     "G205M".Gr.CmdManualOff; // TRAVELLING DRIVE  GERM 6
      S     "G206M".Gr.CmdManualOff; // HORIZONTAL AND LIFTING SCREW  GERM 6
      S     "G209M".Gr.CmdManualOff; // TURNING SCREWS  GERM 6
      S     "G210M".Gr.CmdManualOff; // FAN AND VALVE SRAY AIR  GERM 6
      S     "G211M".Gr.CmdManualOff; // FRESH AIR LOUVER  GERM 6
      S     "G212M".Gr.CmdManualOff; // EXHAUST AIR LOUVER  GERM 6
      S     "G217M".Gr.CmdManualOff; // COOLING / HEATING  GERM 6
//  RESET ADDITIONAL CMD`S
      R     "G202M".USW14; // ILO-cmd
      R     "G202M".USW15; // ILO-cmd
      R     "G203M".USW14; // ILO-cmd
      R     "G203M".USW15; // ILO-cmd
      R     "G204M".USW14; // ILO-cmd
      R     "G204M".USW15; // ILaO-cmd
      R     "G205M".USW14; // ILO-cmd
      R     "G205M".USW15; // ILO-cmd
      R     "G206M".USW14; // ILO-cmd
      R     "G206M".USW15; // ILO-cmd
      R     "G209M".USW14; // ILO-cmd
      R     "G209M".USW15; // ILO-cmd
      R     "G210M".USW14; // ILO-cmd
      R     "G210M".USW15; // ILO-cmd
      R     "G211M".USW14; // ILO-cmd
      R     "G211M".USW15; // ILO-cmd
      R     "G212M".USW14; // ILO-cmd
      R     "G212M".USW15; // ILO-cmd
      R     "G217M".USW14; // ILO-cmd
      R     "G217M".USW15; // ILO-cmd

      U     "MAL1S022".SecAc.Sta1On.Inf08;
      SPB   RSM2;
      L     0;
      T     #tmpInt;
      CALL "SIEMENS_FILL" (
           BVAL                     := #tmpInt,
           RET_VAL                  := #tmpRET,
           BLK                      := "MAL1S022Par".Ilo);
RSM2: NOP   0;


      NOP   0;
// --- FCM 04 - Fans ---
      L     "MAL1S022Par".Ilo.ILOMode;
      L     4;
      <>I   ;
      SPB   IO4;
// man on
      U     "MAL1S022Par".Ilo.GrCMDManOn[1];
      S     "G210M".Gr.InManual; // FAN AND VALVE SRAY AIR  GERM 6
      S     "G211M".Gr.InManual; // FRESH AIR LOUVER  GERM 6
      S     "G212M".Gr.InManual; // EXHAUST AIR LOUVER  GERM 6
      R     "MAL1S022Par".Ilo.GrCMDManOn[1];
// man off
      U     "MAL1S022Par".Ilo.GrCMDManOff[1];
      S     "G210M".Gr.CmdManualOff; // FAN AND VALVE SRAY AIR  GERM 6
      R     "G210M".Gr.InManual; // FAN AND VALVE SRAY AIR  GERM 6
      R     "G210M".USW14; // ILO-cmd
      R     "G210M".USW15; // ILO-cmd
      S     "G211M".Gr.CmdManualOff; // FRESH AIR LOUVER  GERM 6
      R     "G211M".Gr.InManual; // FRESH AIR LOUVER  GERM 6
      R     "G211M".USW14; // ILO-cmd
      R     "G211M".USW15; // ILO-cmd
      S     "G212M".Gr.CmdManualOff; // EXHAUST AIR LOUVER  GERM 6
      R     "G212M".Gr.InManual; // EXHAUST AIR LOUVER  GERM 6
      R     "G212M".USW14; // ILO-cmd
      R     "G212M".USW15; // ILO-cmd
      R     "MAL1S022Par".Ilo.GrCMDManOff[1];
      R     "MAL1S022Par".Ilo.GrCMDManAdditional.Cmd1[1];
      R     "MAL1S022Par".Ilo.GrCMDManAdditional.Cmd2[1];
// man start
      U     "MAL1S022Par".Ilo.GrCMDManStart[1];
      S     "G210M".Gr.CmdOn; // FAN AND VALVE SRAY AIR  GERM 6
      S     "G210M".Gr.CmdContinue; // FAN AND VALVE SRAY AIR  GERM 6
      S     "G211M".Gr.CmdOn; // FRESH AIR LOUVER  GERM 6
      S     "G211M".Gr.CmdContinue; // FRESH AIR LOUVER  GERM 6
      S     "G212M".Gr.CmdOn; // EXHAUST AIR LOUVER  GERM 6
      S     "G212M".Gr.CmdContinue; // EXHAUST AIR LOUVER  GERM 6
      R     "MAL1S022Par".Ilo.GrCMDManStart[1];
      U     "MAL1S022Par".Ilo.GrCMDManStart[2];
      R     "MAL1S022Par".Ilo.GrCMDManStart[2];
// man stop
      U     "MAL1S022Par".Ilo.GrCMDManStop[1];
      S     "G210M".Gr.CmdOff; // FAN AND VALVE SRAY AIR  GERM 6
      S     "G210M".Gr.CmdOff; // FRESH AIR LOUVER  GERM 6
      S     "G210M".Gr.CmdOff; // EXHAUST AIR LOUVER  GERM 6
      R     "MAL1S022Par".Ilo.GrCMDManStop[1];
// man fault reset
      U     "MAL1S022Par".Ilo.GrCMDManOn[17];
      S     "G210M".Gr.CmdFaultReset; // FAN AND VALVE SRAY AIR  GERM 6
      S     "G211M".Gr.CmdFaultReset; // FRESH AIR LOUVER  GERM 6
      S     "G212M".Gr.CmdFaultReset; // EXHAUST AIR LOUVER  GERM 6
      R     "MAL1S022Par".Ilo.GrCMDManOn[17];
// target position
      UN    "G210M".Gr.InManual; // FAN AND VALVE SRAY AIR  GERM 6
      O(    ;
      L     "MAL1S022Par".Ilo.Code_ILO_Funktion0;
      L     400;
      <>I   ;
      )     ;
      SPB   F04a;
      L     "MAL1S022Par".Ilo.SetpointInt01[1];
      T     "MAL1S022Par".Par.ParIntProcess.Speed_ILO_Fan;
F04a: NOP   0;

IO4:  NOP   0;
      NOP   0;
// --- FCM 05 - Fans with target air temperature ---
      L     "MAL1S022Par".Ilo.ILOMode;
      L     5;
      <>I   ;
      SPB   IO5;
// man on
      U     "MAL1S022Par".Ilo.GrCMDManOn[1];
      S     "G210M".Gr.InManual; // FAN AND VALVE SRAY AIR  GERM 6
      S     "G211M".Gr.InManual; // FRESH AIR LOUVER  GERM 6
      S     "G217M".Gr.InManual; // COOLING / HEATING  GERM 6
      R     "MAL1S022Par".Ilo.GrCMDManOn[1];
// man off
      U     "MAL1S022Par".Ilo.GrCMDManOff[1];
      S     "G210M".Gr.CmdManualOff; // FAN AND VALVE SRAY AIR  GERM 6
      R     "G210M".Gr.InManual; // FAN AND VALVE SRAY AIR  GERM 6
      R     "G210M".USW14; // ILO-cmd
      R     "G210M".USW15; // ILO-cmd
      S     "G211M".Gr.CmdManualOff; // FRESH AIR LOUVER  GERM 6
      R     "G211M".Gr.InManual; // FRESH AIR LOUVER  GERM 6
      R     "G211M".USW14; // ILO-cmd
      R     "G211M".USW15; // ILO-cmd
      S     "G217M".Gr.CmdManualOff; // COOLING / HEATING  GERM 6
      R     "G217M".Gr.InManual; // COOLING / HEATING  GERM 6
      R     "G217M".USW14; // ILO-cmd
      R     "G217M".USW15; // ILO-cmd
      R     "MAL1S022Par".Ilo.GrCMDManOff[1];
      R     "MAL1S022Par".Ilo.GrCMDManAdditional.Cmd1[1];
      R     "MAL1S022Par".Ilo.GrCMDManAdditional.Cmd2[1];
// man start
      U     "MAL1S022Par".Ilo.GrCMDManStart[1];
      S     "G210M".Gr.CmdOn; // FAN AND VALVE SRAY AIR  GERM 6
      S     "G210M".Gr.CmdContinue; // FAN AND VALVE SRAY AIR  GERM 6
      S     "G211M".Gr.CmdOn; // FRESH AIR LOUVER  GERM 6
      S     "G211M".Gr.CmdContinue; // FRESH AIR LOUVER  GERM 6
      S     "G217M".Gr.CmdOn; // COOLING / HEATING  GERM 6
      S     "G217M".Gr.CmdContinue; // COOLING / HEATING  GERM 6
      R     "MAL1S022Par".Ilo.GrCMDManStart[1];
      U     "MAL1S022Par".Ilo.GrCMDManStart[2];
      R     "MAL1S022Par".Ilo.GrCMDManStart[2];
// man stop
      U     "MAL1S022Par".Ilo.GrCMDManStop[1];
      S     "G210M".Gr.CmdOff; // FAN AND VALVE SRAY AIR  GERM 6
      S     "G211M".Gr.CmdOff; // FRESH AIR LOUVER  GERM 6
      S     "G217M".Gr.CmdOff; // COOLING / HEATING  GERM 6
      R     "MAL1S022Par".Ilo.GrCMDManStop[1];
// man fault reset
      U     "MAL1S022Par".Ilo.GrCMDManFaultReset[1];
      S     "G210M".Gr.CmdFaultReset; // FAN AND VALVE SRAY AIR  GERM 6
      S     "G211M".Gr.CmdFaultReset; // FRESH AIR LOUVER  GERM 6
      S     "G217M".Gr.CmdFaultReset; // COOLING / HEATING  GERM 6
      R     "MAL1S022Par".Ilo.GrCMDManFaultReset[1];
// target position
      UN    "G217M".Gr.InManual; // COOLING / HEATING  GERM 6
      SPB   F05a;
      L     "MAL1S022Par".Ilo.SetpointInt02[1];
      T     "MAL1S022Par".Par.ParIntProcess.TargetTemperature_ILO;
F05a: NOP   0;
      UN    "G210M".Gr.InManual; // FAN AND VALVE SRAY AIR  GERM 6
      O(    ;
      L     "MAL1S022Par".Ilo.Code_ILO_Funktion0;
      L     500;
      <>I   ;
      )     ;
      SPB   F05b;
      L     "MAL1S022Par".Ilo.SetpointInt01[1];
      T     "MAL1S022Par".Par.ParIntProcess.Speed_ILO_Fan;
F05b: NOP   0;
IO5:  NOP   0;
      NOP   0;
// --- FCM 06 - Fresh air flap ---
      L     "MAL1S022Par".Ilo.ILOMode;
      L     6;
      <>I   ;
      SPB   IO6;
// man on
      U     "MAL1S022Par".Ilo.GrCMDManOn[1];
      S     "G211M".Gr.InManual; // FRESH AIR LOUVER  GERM 6
//      R     DB909.DBX 3032.0
// man off
      U     "MAL1S022Par".Ilo.GrCMDManOff[1];
      S     "G211M".Gr.CmdManualOff; // FRESH AIR LOUVER  GERM 6
      R     "G211M".Gr.InManual; // FRESH AIR LOUVER  GERM 6
      R     "G211M".USW14; // ILO-cmd
      R     "G211M".USW15; // ILO-cmd
      R     "MAL1S022Par".Ilo.GrCMDManOff[1];
      R     "MAL1S022Par".Ilo.GrCMDManAdditional.Cmd1[1];
      R     "MAL1S022Par".Ilo.GrCMDManAdditional.Cmd2[1];
// man start
      U     "MAL1S022Par".Ilo.GrCMDManStart[1];
      S     "G211M".Gr.CmdOn; // FRESH AIR LOUVER  GERM 6
      S     "G211M".Gr.CmdContinue; // FRESH AIR LOUVER  GERM 6
      R     "MAL1S022Par".Ilo.GrCMDManStart[1];
      U     "MAL1S022Par".Ilo.GrCMDManStart[2];
      R     "MAL1S022Par".Ilo.GrCMDManStart[2];

      U     "MAL1S022Par".Ilo.GrCMDManOn[1];
      R     "MAL1S022Par".Ilo.GrCMDManOn[1];
// man stop
      U     "MAL1S022Par".Ilo.GrCMDManStop[1];
      S     "G211M".Gr.CmdOff; // FRESH AIR LOUVER  GERM 6
      R     "MAL1S022Par".Ilo.GrCMDManStop[1];
// man fault reset
      U     "MAL1S022Par".Ilo.GrCMDManOn[17];
      S     "G211M".Gr.CmdFaultReset; // FRESH AIR LOUVER  GERM 6
      R     "MAL1S022Par".Ilo.GrCMDManOn[17];
// moving direction

// target position
      UN    "G211M".Gr.InManual; // FRESH AIR LOUVER  GERM 6
      SPB   F06b;
      L     "MAL1S022Par".Ilo.SetpointInt01[1];
      T     "MAL1S022Par".Par.ParIntProcess.TarPos_ILO_FreshAir;
F06b: NOP   0;

IO6:  NOP   0;
      NOP   0;
// --- FCM 09 - Floor drives ---
      L     "MAL1S022Par".Ilo.ILOMode;
      L     9;
      <>I   ;
      SPB   IO9;
// man on
      U     "MAL1S022Par".Ilo.GrCMDManOn[1];
      S     "G205M".Gr.InManual; // TRAVELLING DRIVE  GERM 6
      S     "G209M".Gr.InManual; // TURNING SCREWS  GERM 6
      R     "MAL1S022Par".Ilo.GrCMDManOn[1];
// man off
      U     "MAL1S022Par".Ilo.GrCMDManOff[1];
      O(    ;
      U(    ;
      U     "G205M".A_2611_BZS44.StTrue; // stop discharge side
      O     "G205M".A_2611_BZS44.InpTrue;
      U     "G205M".Gr.InManual;
      U     "G205M".USW14; // ILO-cmd run fwd
      )     ;
      O(    ;
      U     "G205M".A_2611_BZS46.StTrue; // stop fan side
      O     "G205M".A_2611_BZS46.InpTrue; // stop fan side
      U     "G205M".Gr.InManual;
      U     "G205M".USW15; // ILO-cmd run rev
      )     ;
      U(    ;
      L     "MAL1S022Par".Ilo.ILOMode;
      L     8;
      ==I   ;
      )     ;
      )     ;
      S     "G205M".Gr.CmdManualOff; // TRAVELLING DRIVE  GERM 6
      R     "G205M".Gr.InManual; // TRAVELLING DRIVE  GERM 6
      R     "G205M".USW14; // ILO-cmd
      R     "G205M".USW15; // ILO-cmd
      S     "G209M".Gr.CmdManualOff; // TURNING SCREWS  GERM 6
      R     "G209M".Gr.InManual; // TURNING SCREWS  GERM 6
      R     "G209M".USW14; // ILO-cmd
      R     "G209M".USW15; // ILO-cmd
      R     "MAL1S022Par".Ilo.GrCMDManOff[1];
      R     "MAL1S022Par".Ilo.GrCMDManAdditional.Cmd1[1];
      R     "MAL1S022Par".Ilo.GrCMDManAdditional.Cmd2[1];
// man start
      U     "MAL1S022Par".Ilo.GrCMDManStart[1];
      S     "G205M".Gr.CmdOn; // TRAVELLING DRIVE  GERM 6
      S     "G205M".Gr.CmdContinue; // TRAVELLING DRIVE  GERM 6
      S     "G209M".Gr.CmdOn; // TURNING SCREWS  GERM 6
      S     "G209M".Gr.CmdContinue; // TURNING SCREWS  GERM 6
      U     "MAL1S022Par".Ilo.GrCMDManStart[1];
      R     "MAL1S022Par".Ilo.GrCMDManStart[1];
      U     "MAL1S022Par".Ilo.GrCMDManStart[2];
      R     "MAL1S022Par".Ilo.GrCMDManStart[2];
// man stop
      U     "MAL1S022Par".Ilo.GrCMDManStop[1];
      S     "G205M".Gr.CmdOff; // TRAVELLING DRIVE  GERM 6
      S     "G209M".Gr.CmdOff; // TURNING SCREWS  GERM 6
      R     "MAL1S022Par".Ilo.GrCMDManStop[1];
// man fault reset
      U     "MAL1S022Par".Ilo.GrCMDManFaultReset[1];
      S     "G205M".Gr.CmdFaultReset; // TRAVELLING DRIVE  GERM 6
      S     "G209M".Gr.CmdFaultReset; // TURNING SCREWS  GERM 6
      R     "MAL1S022Par".Ilo.GrCMDManFaultReset[1];
// manual direction
      UN    "G205M".Gr.InManual; // TRAVELLING DRIVE  GERM 6
      SPB   f092;
      U     "MAL1S022Par".Ilo.GrCMDManAdditional.Cmd1[1];
      =     "G205M".USW14; // ILO-cmd run fwd
      U     "MAL1S022Par".Ilo.GrCMDManAdditional.Cmd2[1];
      =     "G205M".USW15; // ILO-cmd run rev
// target position
      L     "MAL1S022Par".Ilo.SetpointInt01[1];
      T     "MAL1S022Par".Par.ParIntProcess.Speed_ILO_FloorRotating;
f092: NOP   0;


IO9:  NOP   0;
// --- FCM 10 - local operating on operating panels ---

      L     "MAL1S022Par".Ilo.ILOMode;
      L     10;
      <>I   ;
      SPB   I10;
// man on
      U     "MAL1S022Par".Ilo.GrCMDManOn[1];
      S     "G205M".Gr.InManual; // Traveling  Drive Germatingbox 6
      S     "G209M".Gr.InManual; // Turning Screws Germinationbox 6
      S     "G204M".Gr.InManual; // Wall locking Germatingbox 6
      S     "G202M".Gr.InManual; // Backwall moving Germatingbox 6
      S     "G203M".Gr.InManual; // Discharger locking Germatingbox 6
      R     "MAL1S022Par".Ilo.GrCMDManOn[1];
// man off
      U     "MAL1S022Par".Ilo.GrCMDManOff[1];
      S     "G205M".Gr.CmdManualOff; // Traveling  Drive Germatingbox 6
      R     "G205M".Gr.InManual; // Traveling  Drive Germatingbox 6
      R     "G205M".USW14; // ILO-cmd
      R     "G205M".USW15; // ILO-cmd
      S     "G209M".Gr.CmdManualOff; // Turning Screws Germinationbox 6
      R     "G209M".Gr.InManual; // Turning Screws Germinationbox 6
      R     "G209M".USW14; // ILO-cmd
      R     "G209M".USW15; // ILO-cmd
      S     "G204M".Gr.CmdManualOff; // Wall locking Germatingbox 6
      R     "G204M".Gr.InManual; // Wall locking Germatingbox 6
      S     "G203M".Gr.CmdManualOff; // Discharger locking Germatingbox 6
      R     "G203M".Gr.InManual; // Discharger locking Germatingbox 6
      S     "G202M".Gr.CmdManualOff; // Backwall moving Germatingbox 6
      R     "G202M".Gr.InManual; // Backwall moving Germatingbox 6
      R     "MAL1S022Par".Ilo.GrCMDManOff[1];
      R     "MAL1S022Par".Ilo.GrCMDManAdditional.Cmd1[1];
      R     "MAL1S022Par".Ilo.GrCMDManAdditional.Cmd2[1];
// man start
      U     "G207M".A_2611_KCL01I1.InpTrue; // pushbutton "start screws"
      S     "G209M".Gr.CmdOn; // Turning Screws Germinationbox 6
      S     "G209M".Gr.CmdContinue; // Turning Screws Germinationbox 6
      S     "G205M".Gr.CmdOn; // Traveling  Drive Germatingbox 6
      S     "G205M".Gr.CmdContinue; // Traveling  Drive Germatingbox 6
      U     "MAL1S022Par".Ilo.GrCMDManStart[1];
      R     "MAL1S022Par".Ilo.GrCMDManStart[1];
      U     "MAL1S022Par".Ilo.GrCMDManStart[2];
      R     "MAL1S022Par".Ilo.GrCMDManStart[2];
// man stop
      UN    "G207M".A_2611_KCL01I2.InpTrue; // pushbutton "stop screws"  //dyk 081025 Inverted
      S     "G209M".Gr.CmdOff; // Turning Screws Germinationbox 6
      U     "MAL1S022Par".Ilo.GrCMDManStop[1];
      O(    ;
      UN    "G207M".A_2611_KCL01I3.InpTrue; // pushbutton "drive fwd"
      UN    "G207M".A_2611_KCL01I4.InpTrue; // pushbutton "drive rev"
      )     ;
      S     "G205M".Gr.CmdOff; // Traveling  Drive Germatingbox 6

      UN    "G204M".Gr.InManual; // Wall locking Germatingbox 6
      O(    ;
      UN    "G207M".A_2615_KCL01I5.InpTrue; // pushbutton "locking"
      UN    "G207M".A_2615_KCL01I6.InpTrue; // pushbutton "unlocking"
      )     ;
      S     "G204M".Gr.CmdOff; // Wall locking/unlocking Germatingbox 6

      UN    "G203M".Gr.InManual; // discharger coupling Germatingbox 6
      O(    ;
      UN    "G207M".A_2615_KCL01I4.InpTrue; // pushbutton "discharger coupling"
      UN    "G207M".A_2615_KCL01I3.InpTrue; // pushbutton "discharger uncoupling"
      )     ;
      S     "G203M".Gr.CmdOff; // discharger coupling Germatingbox 6

      UN    "G202M".Gr.InManual; // Backwall moving Germatingbox 6
      O(    ;
      UN    "G207M".A_2615_KCL01I1.InpTrue; // pushbutton "backwall lifting"
      UN    "G207M".A_2615_KCL01I2.InpTrue; // pushbutton "backwall lowerring"
      )     ;
      S     "G202M".Gr.CmdOff; // Backwall moving Germatingbox 6

      U     "MAL1S022Par".Ilo.GrCMDManStop[1];
      R     "MAL1S022Par".Ilo.GrCMDManStop[1];
// man fault reset
      U     "MAL1S022Par".Ilo.GrCMDManFaultReset[1];
      S     "G205M".Gr.CmdFaultReset; // Traveling  Drive Germatingbox 6
      S     "G209M".Gr.CmdFaultReset; // Turning Screws Germinationbox 6
      R     "MAL1S022Par".Ilo.GrCMDManFaultReset[1];
      NOP   0;
// Manual wall locking
      UN    "G204M".Gr.InManual; // Wall locking Germatingbox 6
      ON    "G207M".A_2615_KCL01I5.InpTrue; // pushbutton "locking"
      SPB   f102;
      S     "G204M".Gr.CmdOn; // Wall locking/unlocking Germatingbox 6
f102: NOP   0;
// Manual wall unlocking
      UN    "G204M".Gr.InManual; // Wall locking Germatingbox 6
      ON    "G207M".A_2615_KCL01I6.InpTrue; // pushbutton "unlocking"
      SPB   f103;
      S     "G204M".Gr.CmdOn; // Wall locking/unlocking Germatingbox 6
f103: NOP   0;
// Manual discharger coupling
      UN    "G203M".Gr.InManual; // discharger coupling Germatingbox 6
      ON    "G207M".A_2615_KCL01I4.InpTrue; // pushbutton "discharger coupling"
      SPB   f104;
      S     "G203M".Gr.CmdOn; // discharger coupling Germatingbox 6
f104: NOP   0;
// Manual discharger uncoupling
      UN    "G203M".Gr.InManual; // discharger coupling Germatingbox 6
      ON    "G207M".A_2615_KCL01I3.InpTrue; // pushbutton "discharger uncoupling"
      SPB   f105;
      S     "G203M".Gr.CmdOn; // discharger coupling Germatingbox 6
f105: NOP   0;
// Manual backwall moving
      UN    "G202M".Gr.InManual; // Backwall moving Germatingbox 6
      ON    "G207M".A_2615_KCL01I1.InpTrue; // pushbutton "backwall lifting"
      SPB   f106;
      S     "G202M".Gr.CmdOn; // Backwall moving Germatingbox 6
f106: NOP   0;
      UN    "G202M".Gr.InManual; // Backwall moving Germatingbox 6
      ON    "G207M".A_2615_KCL01I2.InpTrue; // pushbutton "backwall lowerring"
      SPB   f107;
      S     "G202M".Gr.CmdOn; // Backwall moving Germatingbox 6
f107: NOP   0;
// manual direction
      UN    "G205M".Gr.InManual; // Traveling  Drive Germatingbox 6
      O     ;
      UN    "G207M".A_2611_KCL01I3.InpTrue; // pushbutton "drive fwd"
      UN    "G207M".A_2611_KCL01I4.InpTrue; // pushbutton "drive rev"
      SPB   f109;
      U     "G207M".A_2611_KCL01I3.InpTrue; // pushbutton "drive fwd"
      =     "G205M".USW14; // ILO-cmd run fwd
      S     "G205M".Gr.CmdOn; // Traveling  Drive Germatingbox 6
      U     "G207M".A_2611_KCL01I4.InpTrue; // pushbutton "drive rev"
      =     "G205M".USW15; // ILO-cmd run rev
      S     "G205M".Gr.CmdOn; // Traveling  Drive Germatingbox 6

// target position
      L     "MAL1S022Par".Ilo.SetpointInt01[1];
      T     "MAL1S022Par".Par.ParIntProcess.Speed_ILO_FloorRotating;
f109: NOP   0;

I10:  NOP   0;
//
// copy state
      U     "G205M".Gr.InOutAutostartMan; // TRAVELLING DRIVE  GERM 6
      =     "MAL1S022Par".Ilo.GrSTMan[2];
      U     "G209M".Gr.InOutAutostartMan; // TURNING SCREWS  GERM 6
      =     "MAL1S022Par".Ilo.GrSTMan[6];
      U     "G210M".Gr.InOutAutostartMan; // FAN AND VALVE SRAY AIR  GERM 6
      =     "MAL1S022Par".Ilo.GrSTMan[7];
      U     "G211M".Gr.InOutAutostartMan; // FRESH AIR LOUVER  GERM 6
      =     "MAL1S022Par".Ilo.GrSTMan[8];
      U     "G217M".Gr.InOutAutostartMan; // COOLING / HEATING  GERM 6
      =     "MAL1S022Par".Ilo.GrSTMan[14];

// copy state

NETWORK
TITLE =ASW_9999: Init ASW Flags
// clear all flags explicde to find them back
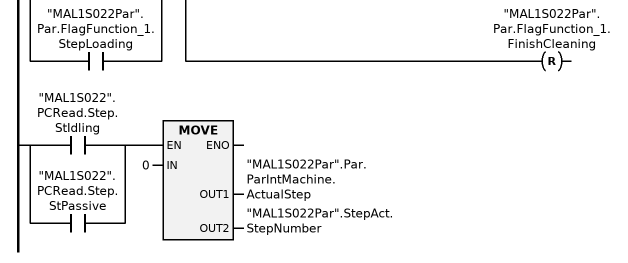
      U     "MAL1S022".PCRead.Step.StIdling;
      O     "MAL1S022".PCRead.Step.StPassive;
      R     "MAL1S022Par".Par.FlagFunction_1.StepLoading;
      R     "MAL1S022Par".Par.FlagFunction_1.StepUnloading;
      R     "MAL1S022Par".Par.FlagFunction_1.StepCleaning;
      R     "MAL1S022Par".Par.FlagFunction_1.LoadingBreak;
      R     "MAL1S022Par".Par.FlagFunction_1.UnloadingBreak;
      R     "MAL1S022Par".Par.FlagFunction_1.CleaningBreak;
      R     "MAL1S022Par".Par.FlagFunction_1.FinishLoading;
      R     "MAL1S022Par".Par.FlagFunction_1.FinishUnloading;
      R     "MAL1S022Par".Par.FlagFunction_1.FinishCleaning;
      R     "MAL1S022Par".Par.FlagFunction_1.Round_1;
      R     "MAL1S022Par".Par.FlagFunction_1.Round_2;
      R     "MAL1S022Par".Par.FlagFunction_1.Round_3;
      R     "MAL1S022Par".Par.FlagFunction_1.Round_4;
      R     "MAL1S022Par".Par.FlagFunction_1.Round_5;
      R     "MAL1S022Par".Par.FlagFunction_1.Round_6;
      R     "MAL1S022Par".Par.FlagFunction_1.Beladung_beendet;
      R     "MAL1S022Par".Par.FlagFunction_1.Entladerunden_erreicht;
      R     "MAL1S022Par".Par.FlagFunction_1.Reinigungsrunde_erreicht;
      R     "MAL1S022Par".Par.FlagGen.TurningStarted;
      R     "MAL1S022Par".Par.FlagFunction_1.TurningStart;
      R     "MAL1S022Par".Par.FlagFunction_1.TurningStop;
      R     "MAL1S022Par".Par.FlagFunction_1.TurningLeft;
      R     "MAL1S022Par".Par.FlagFunction_1.TurningRight;
      R     "MAL1S022Par".Par.FlagFunction_1.LoadFirstPartEnd;
      R     "MAL1S022Par".Par.FlagFunction_1.TurningWithSpraying;
      R     "MAL1S022Par".Par.FlagFunction_1.TurningWithoutSpraying;
      R     "MAL1S022Par".Par.FlagGen.TurningStarted;
      R     "MAL1S022Par".Par.FlagProcess2.Turning1WithoutSpraying;
      R     "MAL1S022Par".Par.FlagProcess2.Turning2WithoutSpraying;
      R     "MAL1S022Par".Par.FlagProcess2.Turning1WithSpraying;
      R     "MAL1S022Par".Par.FlagProcess2.Turning2WithSpraying;
      R     "MAL1S022Par".Par.FlagProcess2.Turning1WithDosing;
      R     "MAL1S022Par".Par.FlagProcess2.Turning2WithDosing;
      R     "MAL1S022Par".Par.FlagProcess2.StartFirstTurningRound;
      R     "MAL1S022Par".Par.FlagProcess2.StartSecondTurningRound;

      R     "MAL1S022Par".Par.FlagFunction_1.UnloadFirstPartEnd;
      R     "MAL1S022Par".Par.FlagFunction_1.UnloadSecondPartEnd;
      R     "MAL1S022Par".Par.FlagFunction_1.UnloadFirstPart;
      R     "MAL1S022Par".Par.FlagFunction_1.UnloadSecondPart;
      R     "MAL1S022Par".Par.FlagFunction_1.UnloadingStarted;
      R     "MAL1S022Par".Par.FlagProcess.ProcessActive;
      R     "MAL1S022Par".Par.FlagProcess.ProcessStartFP;
      R     "MAL1S022Par".Par.FlagProcess.ProcessStartScan;
      R     "MAL1S022Par".Par.FlagProcess.ProcessEnd;
      R     "MAL1S022Par".Par.FlagProcess.FP_SendResultToPIC;
      R     "MAL1S022Par".Par.FlagMachine.ImpulsNullstellung;
      R     "MAL1S022Par".Par.FlagMachine_0.CmdTurnRevAfterUnloading;
      R     "MAL1S022Par".Par.FlagMachine_0.CleaningAfterUnloading;
      R     "MAL1S022Par".Par.FlagMachine_0.CleaningAfterLoading;

//
      U     "MAL1S022".PCRead.Step.StWait;
      O     "MAL1S022Par".Par.FlagFunction_1.StepLoading;
      R     "MAL1S022Par".Par.FlagProcess.ProcessEnd;
      R     "MAL1S022Par".Par.FlagFunction_1.FinishCleaning;

      U     "MAL1S022".PCRead.Step.StIdling;
      O     "MAL1S022".PCRead.Step.StPassive;
      SPBN  csn;
      L     0; // clear step number
      T     "MAL1S022Par".Par.ParIntMachine.ActualStep;
      T     "MAL1S022Par".StepAct.StepNumber;
csn:  NOP   0;

NETWORK
TITLE =Main0_End: Init flag
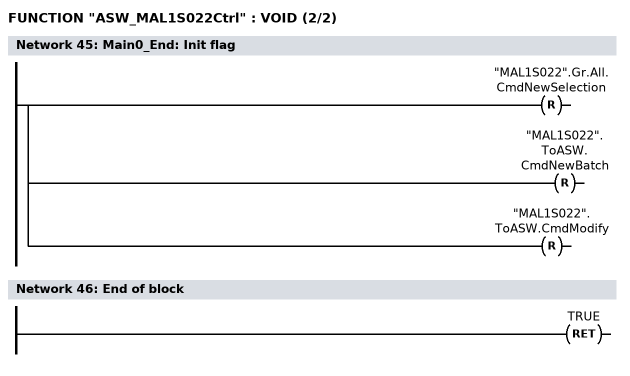

      SET   ;
      R     "MAL1S022".Gr.All.CmdNewSelection;
      R     "MAL1S022".ToASW.CmdNewBatch;
      R     "MAL1S022".ToASW.CmdModify;

NETWORK
TITLE =End of block

      BE    ;

END_FUNCTION

